(* PLC project  *)

CONFIGURATION RaspberryPi_4B
END_CONFIGURATION
